GLOBALCONSTANTS AID_WS (* Working set object attribute ids (all read-only) *)
  (* Standard: 61499-1; Description: Copyright (c) 2023 HR Agrartechnik GmbH This program and the accompanying materials are made available under the terms of the Eclipse Public License 2.0 which is available at https://www.eclipse.org/legal/epl-2.0/ SPDX-License-Identifier: EPL-2.0 *)
  (* Version 1.0, 2026-06-20, Franz Höpfinger, HR Agrartechnik GmbH *)
  PACKAGE isobus::UT::Q::const::AID;
  VAR_GLOBAL CONSTANT
    BACKGROUND_COLOUR : USINT := USINT#1; (* 1: AID_WS_BACKGROUND_COLOUR (read-only) - Background colour index. *)
    SELECTABLE : USINT := USINT#2; (* 2: AID_WS_SELECTABLE (read-only) - 0 = FALSE, 1 = TRUE. Indicates whether or not this Working Set can be *)
    ACTIVE_MASK : USINT := USINT#3; (* 3: AID_WS_ACTIVE_MASK (read-only) - The Object ID of the Data or Alarm Mask to display whenever the Working Set is active. Query via Get Attribute Value (F.58); modify via Change Active Mask (F.34). *)
  END_VAR
END_GLOBALCONSTANTS
